FUNCTION Height_To_Anology : INT
VAR_INPUT
	height	:REAL;
END_VAR
VAR
	i,j	:INT;
	rtn :INT;
END_VAR

i:=TO_INT(height*10)/10;
j:=TO_INT(height*10) MOD 10;


rtn:=(HeightMap[i+1]-HeightMap[i])*j/10 + HeightMap[i];


Height_To_Anology:=rtn;

END_FUNCTION

(* stored: Version 1.1.0.1, ProductVersion 3.1.4024.12
   POU Height_To_Anology: Id {43a6637c-aba7-421b-af8d-b1cab85240b0}, SpecialFunc None *)
